Universal Robots PolyScope program: BiBaZu_GUI.urp

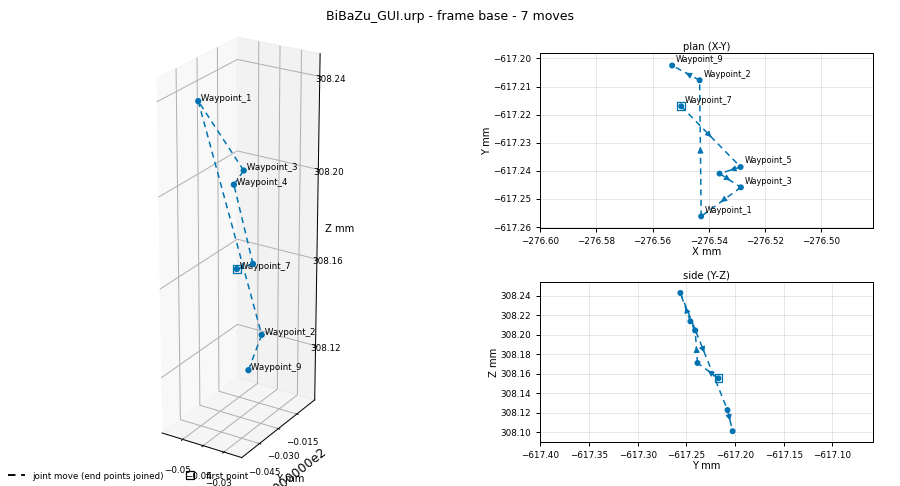
[picture p0: tool path of BiBaZu_GUI.urp in frame base, 7 of 7 moves have a stored position in this frame; points joined in program order, loops and branches not executed]
Program BiBaZu_GUI (installation=default directory=/programs/usbdisk createdIn=5.12.3.1101619 lastSavedIn=5.12.3.1101619 robotSerialNumber=20225600150)
Calibrated DH parameters: a=[0.000094, -0.358471, -0.354967, -0.000026, 0.000038, 0]; d=[0.180831, -2593.499827, 2607.523833, -13.849973, 0.119817, 0.115619]; alpha=[1.570306, -0.000122, 0.004332, 1.569125, -1.569785, 0]; deltaTheta=[0, 0.723437, 5.729253, -0.169511, 0.000001, 0]
BeforeStart
  Script file BiBaZu_GUI_Init.script
    | def BiBaZu_GUI_Init():
    |   global angle = 0
    |   global last_command = read_input_integer_register(43)
    |   global active_command = last_command
    |   global command_valid = False
    |   write_output_integer_register(42, last_command)
    |   write_output_integer_register(43, 1)
    |   write_output_integer_register(41, 0)
    | end
    | 
    | BiBaZu_GUI_Init()
Robot Program (runOnlyOnce=false)
  angle := 0
  Script file BiBaZu_GUI_Wait.script
    | def BiBaZu_GUI_Wait():
    |   local command = read_input_integer_register(43)
    |   while command == last_command:
    |     sync()
    |     command = read_input_integer_register(43)
    |   end
    | 
    |   local requested_angle = read_input_integer_register(42)
    |   local valid = requested_angle == 155 or requested_angle == 160 or requested_angle == 170 or requested_angle == 180 or requested_angle == 190 or requested_angle == 200 or requested_angle == 210
    | 
    |   if valid:
    |     global angle = requested_angle
    |     global active_command = command
    |     global command_valid = True
    |     write_output_integer_register(43, 2)
    |   else:
    |     global angle = 0
    |     global command_valid = False
    |     global last_command = command
    |     write_output_integer_register(43, -1)
    |     write_output_integer_register(42, command)
    |   end
    | end
    | 
    | BiBaZu_GUI_Wait()
  Switch expression=angle
    Case (caseValue=155)
      MoveJ speed 60 deg/s, acceleration 80 deg/s^2 (useActiveTCP=true) feature=Base
        Waypoint Waypoint_7: TCP in base x=-276.55 y=-617.217 z=308.155 mm, rx=0.3791 ry=1.154 rz=-2.785 rad; joints [-98.343, -121.404, -107.869, 272.447, -84.891, -162.969] deg
    Case (caseValue=160)
      MoveJ speed 60 deg/s, acceleration 80 deg/s^2 (useActiveTCP=true) feature=Base
        Waypoint Waypoint_5: TCP in base x=-276.529 y=-617.239 z=308.171 mm, rx=0.3908 ry=1.1522 rz=-2.7805 rad; joints [-98.271, -121.358, -107.877, 272.307, -84.501, -162.652] deg
    Case (caseValue=170)
      MoveJ speed 60 deg/s, acceleration 80 deg/s^2 (useActiveTCP=true) feature=Base
        Waypoint Waypoint_4: TCP in base x=-276.536 y=-617.241 z=308.204 mm, rx=0.4142 ry=1.1483 rz=-2.7715 rad; joints [-98.135, -121.265, -107.892, 272.028, -83.726, -162.018] deg
    Case (caseValue=180)
      MoveJ speed 60 deg/s, acceleration 80 deg/s^2 (useActiveTCP=true) feature=Base
        Waypoint Waypoint_3: TCP in base x=-276.529 y=-617.246 z=308.214 mm, rx=0.4375 ry=1.1444 rz=-2.7623 rad; joints [-97.997, -121.173, -107.904, 271.738, -82.953, -161.379] deg
    Case (caseValue=190)
      MoveJ speed 60 deg/s, acceleration 80 deg/s^2 (useActiveTCP=true) feature=Base
        Waypoint Waypoint_1: TCP in base x=-276.543 y=-617.256 z=308.243 mm, rx=0.4607 ry=1.1404 rz=-2.753 rad; joints [-97.862, -121.079, -107.908, 271.432, -82.182, -160.736] deg
    Case (caseValue=200)
      MoveJ speed 60 deg/s, acceleration 80 deg/s^2 (useActiveTCP=true) feature=Base
        Waypoint Waypoint_2: TCP in base x=-276.543 y=-617.208 z=308.123 mm, rx=0.4838 ry=1.1369 rz=-2.7432 rad; joints [-97.727, -120.986, -107.921, 271.106, -81.419, -160.085] deg
    Case (caseValue=210)
      MoveJ speed 60 deg/s, acceleration 80 deg/s^2 (useActiveTCP=true) feature=Base
        Waypoint Waypoint_9: TCP in base x=-276.553 y=-617.203 z=308.101 mm, rx=0.5068 ry=1.1329 rz=-2.7336 rad; joints [-97.593, -120.891, -107.92, 270.774, -80.654, -159.434] deg
  Script file BiBaZu_GUI_Ack.script
    | def BiBaZu_GUI_Ack():
    |   if command_valid:
    |     write_output_integer_register(41, angle)
    |     write_output_integer_register(43, 3)
    |     write_output_integer_register(42, active_command)
    |     global last_command = active_command
    |     global command_valid = False
    |   end
    | end
    | 
    | BiBaZu_GUI_Ack()
